// TIA Portal V19 export
DATA_BLOCK "FAULTS"   // DB14
{ S7_Optimized_Access := 'FALSE' }
   VAR
      ADIN { S7_SetPoint := 'True'} : Array[0.."MAX_ADIN"] of "UDT_DINFAULTS";   // ADIN = 1 alarm/instance, 24 x 8 (each type contains 8 instances) = 192 alarms, offset = 0
      AIN { S7_SetPoint := 'True'} : Array[0.."MAX_AIN"] of "UDT_AINFAULTS";   // AIN = 2 alarms/instance, 200 x 2 = 400 alarms, offset = 192
      DIFF { S7_SetPoint := 'True'} : Array[0.."MAX_DIFF"] of "UDT_AINFAULTS";   // DIFF = 2 alarms/instance, 32 x 2 = 64 alarms, offset = 592
      DIN { S7_SetPoint := 'True'} : Array[0.."MAX_DIN"] of "UDT_DINFAULTS";   // DIN = 1 alarm/instance, 24 x 8 (each type contains 8 instances) = 192 alarms, offset = 656
      MTR { S7_SetPoint := 'True'} : Array[0.."MAX_MTR"] of "UDT_MTRFAULTS";   // MTR = 6 alarms/instance, 200 x 6 = 1200 alarms, offset = 848
      MTRLIN { S7_SetPoint := 'True'} : Array[0.."MAX_MTRLIN"] of "UDT_MTRFAULTS";   // MTRLIN = 6 alarms/instance, 80 x 6 = 480 alarms, offset = 2048
      MTRDIR { S7_SetPoint := 'True'} : Array[0.."MAX_MTRDIR"] of "UDT_MTRFAULTS";   // MTRDIR = 6 alarms/instance, 200 x 6 = 1200 alarms, offset = 2528
      VLV { S7_SetPoint := 'True'} : Array[0.."MAX_VLV"] of "UDT_VALVEFAULTS";   // VLV = 4 alarms/instance, 200 x 6 = 1200 alarms, offset = 3728
      Plant { S7_SetPoint := 'True'} : Array[0.."MAX_PLANT"] of "UDT_DINFAULTS";   // Plant = 1 alarm/instance, 24 x 8 (each type contains 8 instances) = 192 alarms, offset = 4928
   END_VAR
BEGIN
END_DATA_BLOCK
